type ST_Syntax_Bitfields :
struct
    bBit0 : bit;
    bBit1 : bit;
    bBit2 : bit;
    bBit3 : bit;
    nPadding : byte;
end_struct
end_type

(* stored: Version 1.1.0.1, ProductVersion 3.1.4024.16
   DUT ST_Syntax_Bitfields: Id {114239da-90a7-44ca-9d3e-d9984b8f1425} *)
